// TIA Portal V18 export
// export: Created 2026-01-09T11:31:57.2261473Z, ExportSetting WithDefaults, DisplayName Totally Integrated Automation Portal, DisplayVersion V18 Update 5, DisplayName TIA Portal Openness, DisplayVersion V18 Update 5, DisplayName TIA Portal Teamcenter Gateway, DisplayVersion V18, DisplayName TIA Portal Version Control Interface, DisplayVersion V18, DisplayName SINAMICS Startdrive Advanced, DisplayVersion V18 SP2 Update 1, DisplayName SINAMICS Startdrive G110M, G120, G120C, G120D, G120P, G115D, DisplayVersion V18 SP2 Update 1, DisplayName SINAMICS Startdrive G130, G150, S120, S150, SINAMICS MV, S210, G220, S200, DisplayVersion V18 SP2 Update 1, DisplayName STEP 7 Professional, DisplayVersion V18 Update 5, DisplayName STEP 7 Safety, DisplayVersion V18, DisplayName WinCC Professional, DisplayVersion V18 Update 5
TagTable "ST350_FixtureCheck"
  STxxx_GeneralData_FixtureIDCheck{1} : FixtureCheck_UDT  (PLC tag ST10_GeneralData.FixtureIDCheck[1], CPU S71500-2PN_TP700, 1 s)
    TagStructureMember "FixtureIDSetValue"
    TagStructureMember "FixtureIDCheckValue"
    TagStructureMember "FixtureCheckResult"
    TagStructureMember "FixtureCheckUnEnable"
  STxxx_GeneralData_FixtureIDCheck{2} : FixtureCheck_UDT  (PLC tag ST10_GeneralData.FixtureIDCheck[2], CPU S71500-2PN_TP700, 1 s)
    TagStructureMember "FixtureIDSetValue"
    TagStructureMember "FixtureIDCheckValue"
    TagStructureMember "FixtureCheckResult"
    TagStructureMember "FixtureCheckUnEnable"
  STxxx_GeneralData_FixtureIDCheck{3} : FixtureCheck_UDT  (PLC tag ST10_GeneralData.FixtureIDCheck[3], CPU S71500-2PN_TP700, 1 s)
    TagStructureMember "FixtureIDSetValue"
    TagStructureMember "FixtureIDCheckValue"
    TagStructureMember "FixtureCheckResult"
    TagStructureMember "FixtureCheckUnEnable"
  STxxx_GeneralData_FixtureIDCheck{4} : FixtureCheck_UDT  (PLC tag ST10_GeneralData.FixtureIDCheck[4], CPU S71500-2PN_TP700, 1 s)
    TagStructureMember "FixtureIDSetValue"
    TagStructureMember "FixtureIDCheckValue"
    TagStructureMember "FixtureCheckResult"
    TagStructureMember "FixtureCheckUnEnable"
  STxxx_GeneralData_FixtureIDCheck{5} : FixtureCheck_UDT  (PLC tag ST10_GeneralData.FixtureIDCheck[5], CPU S71500-2PN_TP700, 1 s)
    TagStructureMember "FixtureIDSetValue"
    TagStructureMember "FixtureIDCheckValue"
    TagStructureMember "FixtureCheckResult"
    TagStructureMember "FixtureCheckUnEnable"
  STxxx_GeneralData_FixtureIDCheck{6} : FixtureCheck_UDT  (PLC tag ST10_GeneralData.FixtureIDCheck[6], CPU S71500-2PN_TP700, 1 s)
    TagStructureMember "FixtureIDSetValue"
    TagStructureMember "FixtureIDCheckValue"
    TagStructureMember "FixtureCheckResult"
    TagStructureMember "FixtureCheckUnEnable"
  STxxx_GeneralData_FixtureIDCheck{7} : FixtureCheck_UDT  (PLC tag ST10_GeneralData.FixtureIDCheck[7], CPU S71500-2PN_TP700, 1 s)
    TagStructureMember "FixtureIDSetValue"
    TagStructureMember "FixtureIDCheckValue"
    TagStructureMember "FixtureCheckResult"
    TagStructureMember "FixtureCheckUnEnable"
  STxxx_GeneralData_FixtureIDCheck{8} : FixtureCheck_UDT  (PLC tag ST10_GeneralData.FixtureIDCheck[8], CPU S71500-2PN_TP700, 1 s)
    TagStructureMember "FixtureIDSetValue"
    TagStructureMember "FixtureIDCheckValue"
    TagStructureMember "FixtureCheckResult"
    TagStructureMember "FixtureCheckUnEnable"
  STxxx_GeneralData_FixtureIDCheck{9} : FixtureCheck_UDT  (PLC tag ST10_GeneralData.FixtureIDCheck[9], CPU S71500-2PN_TP700, 1 s)
    TagStructureMember "FixtureIDSetValue"
    TagStructureMember "FixtureIDCheckValue"
    TagStructureMember "FixtureCheckResult"
    TagStructureMember "FixtureCheckUnEnable"
  STxxx_GeneralData_FixtureIDCheck{10} : FixtureCheck_UDT  (PLC tag ST10_GeneralData.FixtureIDCheck[10], CPU S71500-2PN_TP700, 1 s)
    TagStructureMember "FixtureIDSetValue"
    TagStructureMember "FixtureIDCheckValue"
    TagStructureMember "FixtureCheckResult"
    TagStructureMember "FixtureCheckUnEnable"
  STxxx_GeneralData_FixtureIDCheck{11} : FixtureCheck_UDT  (PLC tag ST10_GeneralData.FixtureIDCheck[11], CPU S71500-2PN_TP700, 1 s)
    TagStructureMember "FixtureIDSetValue"
    TagStructureMember "FixtureIDCheckValue"
    TagStructureMember "FixtureCheckResult"
    TagStructureMember "FixtureCheckUnEnable"
  STxxx_GeneralData_FixtureIDCheck{12} : FixtureCheck_UDT  (PLC tag ST10_GeneralData.FixtureIDCheck[12], CPU S71500-2PN_TP700, 1 s)
    TagStructureMember "FixtureIDSetValue"
    TagStructureMember "FixtureIDCheckValue"
    TagStructureMember "FixtureCheckResult"
    TagStructureMember "FixtureCheckUnEnable"
  STxxx_GeneralData_FixtureIDCheck{13} : FixtureCheck_UDT  (PLC tag ST10_GeneralData.FixtureIDCheck[13], CPU S71500-2PN_TP700, 1 s)
    TagStructureMember "FixtureIDSetValue"
    TagStructureMember "FixtureIDCheckValue"
    TagStructureMember "FixtureCheckResult"
    TagStructureMember "FixtureCheckUnEnable"
  STxxx_GeneralData_FixtureIDCheck{14} : FixtureCheck_UDT  (PLC tag ST10_GeneralData.FixtureIDCheck[14], CPU S71500-2PN_TP700, 1 s)
    TagStructureMember "FixtureIDSetValue"
    TagStructureMember "FixtureIDCheckValue"
    TagStructureMember "FixtureCheckResult"
    TagStructureMember "FixtureCheckUnEnable"
  STxxx_GeneralData_FixtureIDCheck{15} : FixtureCheck_UDT  (PLC tag ST10_GeneralData.FixtureIDCheck[15], CPU S71500-2PN_TP700, 1 s)
    TagStructureMember "FixtureIDSetValue"
    TagStructureMember "FixtureIDCheckValue"
    TagStructureMember "FixtureCheckResult"
    TagStructureMember "FixtureCheckUnEnable"
  STxxx_GeneralData_FixtureIDCheck{16} : FixtureCheck_UDT  (PLC tag ST10_GeneralData.FixtureIDCheck[16], CPU S71500-2PN_TP700, 1 s)
    TagStructureMember "FixtureIDSetValue"
    TagStructureMember "FixtureIDCheckValue"
    TagStructureMember "FixtureCheckResult"
    TagStructureMember "FixtureCheckUnEnable"
